(* IEC 61131-3 sources: ironplc-benchmarks/benchmarks/programs, 13 files *)

(* ---- arithmetic.st ---- *)
(* arithmetic.st — Integer arithmetic operations.
   Exercises ADD, SUB, MUL, DIV, and MOD with analytically verifiable
   outputs. After each cycle, result_add = 30, result_sub = 10,
   result_mul = 200, result_div = 2, result_mod = 0. *)

PROGRAM arithmetic
VAR
    a : INT := 20;
    b : INT := 10;
    result_add : INT;
    result_sub : INT;
    result_mul : INT;
    result_div : INT;
    result_mod : INT;
END_VAR
    result_add := a + b;
    result_sub := a - b;
    result_mul := a * b;
    result_div := a / b;
    result_mod := a MOD b;
END_PROGRAM

(* ---- blinky.st ---- *)
(* blinky.st — Minimal benchmark baseline.
   Toggles an output coil on each scan cycle. Exercises the absolute
   minimum VM path: variable read, boolean NOT, variable write. *)

PROGRAM blinky
VAR
    output : BOOL := FALSE;
END_VAR
    output := NOT output;
END_PROGRAM

(* ---- case_state.st ---- *)
(* case_state.st — CASE-based state machine.
   Cycles through 4 states on each scan. Exercises CASE/branch opcodes
   which map to jump tables in both compiled and interpreted execution. *)

PROGRAM case_state
VAR
    state : INT := 0;
    output_a : BOOL := FALSE;
    output_b : BOOL := FALSE;
    output_c : BOOL := FALSE;
    output_d : BOOL := FALSE;
END_VAR
    CASE state OF
        0:
            output_a := TRUE;
            output_b := FALSE;
            output_c := FALSE;
            output_d := FALSE;
            state := 1;
        1:
            output_a := FALSE;
            output_b := TRUE;
            output_c := FALSE;
            output_d := FALSE;
            state := 2;
        2:
            output_a := FALSE;
            output_b := FALSE;
            output_c := TRUE;
            output_d := FALSE;
            state := 3;
        3:
            output_a := FALSE;
            output_b := FALSE;
            output_c := FALSE;
            output_d := TRUE;
            state := 0;
    END_CASE;
END_PROGRAM

(* ---- counter_up.st ---- *)
(* counter_up.st — Counter with reset.
   Exercises integer arithmetic, comparison, and conditional assignment.
   The counter increments each cycle and resets at a threshold. *)

PROGRAM counter_up
VAR
    count : INT := 0;
    threshold : INT := 1000;
    reset_flag : BOOL := FALSE;
END_VAR
    IF count >= threshold THEN
        count := 0;
        reset_flag := TRUE;
    ELSE
        count := count + 1;
        reset_flag := FALSE;
    END_IF;
END_PROGRAM

(* ---- for_loop.st ---- *)
(* for_loop.st — FOR loop with accumulator.
   Exercises loop control flow opcodes. Sums integers 1..100 each cycle,
   producing a verifiable result of 5050. *)

PROGRAM for_loop
VAR
    i : INT;
    total : INT := 0;
END_VAR
    total := 0;
    FOR i := 1 TO 100 DO
        total := total + i;
    END_FOR;
END_PROGRAM

(* ---- oscat_binom.st ---- *)
(* oscat_binom.st — Binomial coefficient from OSCAT library.
   Source: https://github.com/PLC-lang/oscat (OSCAT BASIC, www.oscat.de)
   Exercises: FOR loop, IF/ELSIF/ELSE, RETURN, integer multiply/divide.
   BINOM(10, 5) = 252 each cycle. *)

FUNCTION BINOM : DINT
VAR_INPUT
	N : INT;
	K : INT;
END_VAR
VAR
	i: INT;
END_VAR
(* @END_DECLARATION := '0' *)
IF 2 * K > n THEN
	k := n - k;
END_IF;
IF k > n THEN
	RETURN;
ELSIF k = 0 OR k = n THEN
	BINOM := 1;
ELSIF k = 1 THEN
	BINOM := n;
ELSE
	BINOM := n;
	n := n + 1;
	FOR i := 2 TO k DO
		BINOM := BINOM * (n - i) / i;
	END_FOR;
END_IF;
END_FUNCTION

PROGRAM oscat_binom
VAR
    result : INT;
END_VAR
    result := DINT_TO_INT(BINOM(N := 10, K := 5));
END_PROGRAM

(* ---- oscat_expn.st ---- *)
(* oscat_expn.st — Fast integer exponentiation by squaring from OSCAT.
   Source: https://github.com/PLC-lang/oscat (OSCAT BASIC, www.oscat.de)
   Exercises: WHILE loop, bit access (.0, .15), SHR, REAL arithmetic.
   EXPN(2.0, 10) = 1024.0 each cycle. *)

FUNCTION EXPN : REAL
VAR_INPUT
	X : REAL;
	N : INT;
END_VAR
VAR
	sign: BOOL;
END_VAR
(* @END_DECLARATION := '0' *)
sign := n.15;
N := ABS(N);
IF N.0 THEN EXPN := X; ELSE EXPN := 1.0; END_IF;
N := SHR(N,1);
WHILE N > 0 DO
   X := X * X;
   IF N.0 THEN EXPN := EXPN * X; END_IF;
   N := SHR(N,1);
END_WHILE;
IF sign THEN EXPN := 1.0 / EXPN; END_IF;
END_FUNCTION

PROGRAM oscat_expn
VAR
    result : INT;
END_VAR
    result := REAL_TO_INT(EXPN(X := 2.0, N := 10));
END_PROGRAM

(* ---- oscat_fib.st ---- *)
(* oscat_fib.st — Fibonacci sequence from OSCAT library.
   Source: https://github.com/PLC-lang/oscat (OSCAT BASIC, www.oscat.de)
   Exercises: WHILE loop, IF/ELSIF/ELSE, RETURN, integer arithmetic.
   FIB(20) = 6765 each cycle. *)

FUNCTION FIB : DINT
VAR_INPUT
	X : INT;
END_VAR
VAR
	t1, t2: DINT;
END_VAR
(* @END_DECLARATION := '0' *)
IF X < 0 OR X > 46 THEN
	FIB := -1;
ELSIF x < 2 THEN
	FIB := X;
	RETURN;
ELSE
	t2 := 1;
	WHILE X > 3 DO
		X := X-2;
		t1 := t1 + t2;
		t2 := t1 + t2;
	END_WHILE;
	IF X > 2 THEN t1 := t1 + t2; END_IF;
	fib := t1 + t2;
END_IF;
END_FUNCTION

PROGRAM oscat_fib
VAR
    result : INT;
END_VAR
    result := DINT_TO_INT(FIB(X := 20));
END_PROGRAM

(* ---- oscat_gcd.st ---- *)
(* oscat_gcd.st — Greatest common divisor (Stein's binary algorithm) from OSCAT.
   Source: https://github.com/PLC-lang/oscat (OSCAT BASIC, www.oscat.de)
   Exercises: nested WHILE loops, bit access (.0), SHR/SHL, ABS.
   GCD(48, 36) = 12 each cycle. *)

FUNCTION GCD : INT
VAR_INPUT
	A : DINT;
	B : DINT;
END_VAR
VAR
	t: DINT;
END_VAR
(* @END_DECLARATION := '0' *)
IF A = 0 THEN
	GCD := DINT_TO_INT(ABS(B));
ELSIF B = 0 THEN
	GCD := DINT_TO_INT(ABS(A));
ELSE
	A := ABS(A);
	B := ABS(B);
	GCD := 1;
	WHILE NOT(A.0 OR B.0) DO
		A := SHR(A,1);
		B := SHR(B,1);
		GCD := SHL(GCD,1);
	END_WHILE;
	WHILE A > 0 DO
		IF NOT(A.0) THEN A := SHR(A,1);
		ELSIF NOT(B.0) THEN B := SHR(B,1);
		ELSE
			t:= SHR(ABS(A-B),1);
			IF A < B THEN B := t; ELSE A := T; END_IF;
		END_IF;
	END_WHILE;
	GCD := GCD * DINT_TO_INT(B);
END_IF;
END_FUNCTION

PROGRAM oscat_gcd
VAR
    result : INT;
END_VAR
    result := GCD(A := 48, B := 36);
END_PROGRAM

(* ---- oscat_lambert_w.st ---- *)
(* oscat_lambert_w.st — Lambert W function from OSCAT.
   Source: https://github.com/PLC-lang/oscat (OSCAT BASIC, www.oscat.de)
   Exercises: FOR loop with EXIT, EXP, LN, REAL arithmetic, RETURN,
   IF/ELSIF/ELSE, REAL_TO_DW (bitwise float comparison via REF_TO).
   LAMBERT_W(1.0) ~= 0.5671 each cycle, result = 5671. *)

FUNCTION REAL_TO_DW : DWORD
VAR_INPUT
	X : REAL;
END_VAR
VAR
	pt : REF_TO DWORD;
END_VAR
(* @END_DECLARATION := '0' *)
pt := REF(X);
REAL_TO_DW := pt^;
END_FUNCTION

FUNCTION LAMBERT_W : REAL
VAR_INPUT
	X : REAL;
END_VAR
VAR
	w : REAL;
	i : INT;
	we: REAL;
	w1e: REAL;
	last: DWORD;
	ewx: REAL;
END_VAR
(* @END_DECLARATION := '0' *)
IF x < -0.367879441171442 THEN
	LAMBERT_W := -1000.0;
	RETURN;
ELSIF x = 0.0 THEN
	RETURN;
ELSIF x <= 500.0 THEN
	w := LN(x + 1.0);
	w := 0.665 * (1.0 + 0.0195 * w) * w + 0.04;
ELSE
	w := LN(x - 4.0) - (1.0 - 1.0/LN(x)) * LN(LN(x));
END_IF;
FOR i := 0 TO 5 DO
	ewx := EXP(w);
	we := w * ewx - x;
	w1e := (w+1.0) * ewx;
	last := REAL_TO_DW(w) AND 16#FFFF_FFFC;
	w := w - (we / (w1e - (w+2.0) * we / (2.0 * w + 2.0)));
	IF (REAL_TO_DW(w) AND 16#FFFF_FFFC) = last THEN EXIT; END_IF;
END_FOR;
LAMBERT_W := w;
END_FUNCTION

PROGRAM oscat_lambert_w
VAR
    result : INT;
END_VAR
    result := REAL_TO_INT(LAMBERT_W(X := 1.0) * 10000.0);
END_PROGRAM

(* ---- oscat_linear_int.st ---- *)
(* oscat_linear_int.st — Piecewise linear interpolation from OSCAT.
   Source: https://github.com/PLC-lang/oscat (OSCAT BASIC, www.oscat.de)
   Exercises: WHILE loop, 2D array access, REAL arithmetic, MIN.
   Interpolates X=25 over 5 points: (0,0),(10,100),(20,200),(30,300),(40,400).
   Result = 250 each cycle. *)

FUNCTION LINEAR_INT : REAL
VAR_INPUT
	X : REAL;
	XY : ARRAY[1..20,0..1] OF REAL;
	Pts : INT;
END_VAR
VAR
	i : INT;
END_VAR
(* @END_DECLARATION := '0' *)
pts := MIN(pts,20);

i := 2;
WHILE (i < pts) AND (XY[i,0] < X) DO
	i := i + 1;
END_WHILE;

LINEAR_INT := ((XY[i,1] - XY[i-1,1]) * X - XY[i,1] * XY[i-1,0] + XY[i-1,1] * XY[i,0]) / (XY[i,0] - XY[i-1,0]);
END_FUNCTION

PROGRAM oscat_linear_int
VAR
    points : ARRAY[1..20,0..1] OF REAL;
    result : INT;
END_VAR
    points[1,0] := 0.0;   points[1,1] := 0.0;
    points[2,0] := 10.0;  points[2,1] := 100.0;
    points[3,0] := 20.0;  points[3,1] := 200.0;
    points[4,0] := 30.0;  points[4,1] := 300.0;
    points[5,0] := 40.0;  points[5,1] := 400.0;
    result := REAL_TO_INT(LINEAR_INT(X := 25.0, XY := points, Pts := 5));
END_PROGRAM

(* ---- oscat_polynom_int.st ---- *)
(* oscat_polynom_int.st — Newton polynomial interpolation from OSCAT.
   Source: https://github.com/PLC-lang/oscat (OSCAT BASIC, www.oscat.de)
   Exercises: nested FOR loops (BY -1), 2D array access, REAL arithmetic, MIN.
   Interpolates X=2.5 over y=x^2 points: (1,1),(2,4),(3,9),(4,16),(5,25).
   Result = REAL_TO_INT(6.25) = 6 each cycle. *)

FUNCTION POLYNOM_INT : REAL
VAR_INPUT
	X : REAL;
	XY : ARRAY[1..5,0..1] OF REAL;
	Pts : INT;
END_VAR
VAR
	I, J : INT;
	stop: INT;
END_VAR
(* @END_DECLARATION := '0' *)
pts := MIN(pts, 5);

FOR i := 1 TO pts DO
	stop := i + 1;
   	FOR j := pts TO stop BY -1 DO
   		XY[j,1] := (XY[j,1] - XY[j-1,1]) / (XY[j,0] - XY[j-i,0]);
	END_FOR;
END_FOR;

POLYNOM_INT := 0.0;
FOR i := pts TO 1 BY -1 DO
       POLYNOM_INT := POLYNOM_INT * (X - XY[i,0]) + XY[i,1];
END_FOR;
END_FUNCTION

PROGRAM oscat_polynom_int
VAR
    points : ARRAY[1..5,0..1] OF REAL;
    result : INT;
END_VAR
    points[1,0] := 1.0;  points[1,1] := 1.0;
    points[2,0] := 2.0;  points[2,1] := 4.0;
    points[3,0] := 3.0;  points[3,1] := 9.0;
    points[4,0] := 4.0;  points[4,1] := 16.0;
    points[5,0] := 5.0;  points[5,1] := 25.0;
    result := REAL_TO_INT(POLYNOM_INT(X := 2.5, XY := points, Pts := 5));
END_PROGRAM

(* ---- oscat_real_to_frac.st ---- *)
(* oscat_real_to_frac.st — Real to fraction (continued fractions) from OSCAT.
   Source: https://github.com/PLC-lang/oscat (OSCAT BASIC, www.oscat.de)
   Exercises: REPEAT/UNTIL loop, EXIT, IF/ELSE, REAL/DINT arithmetic,
   struct return type, ABS, type conversions.
   REAL_TO_FRAC(3.14159, 1000) = 355/113 each cycle. *)

TYPE FRACTION :
STRUCT
	NUMERATOR : INT;
	DENOMINATOR : INT;
END_STRUCT
END_TYPE

FUNCTION REAL_TO_FRAC : FRACTION
VAR_INPUT
	X : REAL;
	N : INT;
END_VAR
VAR
	temp : DINT;
	sign: BOOL;
	X_gerundet: DINT;
	X_ohne_Nachkomma: REAL;
	Numerator:       DINT := 1;
	Denominator:     DINT := 0;
	Numerator_old:   DINT := 0;
	Denominator_old: DINT := 1;
END_VAR
(* @END_DECLARATION := '0' *)
IF X < 0.0 THEN
	sign := TRUE;
	X := ABS(X);
END_IF;

REPEAT
	X_gerundet := REAL_TO_DINT(X);

	temp := numerator * X_gerundet + numerator_old;
	numerator_old := numerator;
	numerator := temp;

	temp := denominator * X_gerundet + denominator_old;
	denominator_old := denominator;
	denominator := temp;

	X_ohne_Nachkomma := DINT_TO_REAL(X_gerundet);
	IF X = X_ohne_Nachkomma THEN
		IF ABS(denominator) <= N THEN
			numerator_old := numerator;
			denominator_old := denominator;
		END_IF;
		EXIT;
	ELSE
		X := 1.0 / (X - X_ohne_Nachkomma);
	END_IF;

UNTIL
	ABS(Denominator) > N
END_REPEAT;

IF sign THEN
	REAL_TO_FRAC.NUMERATOR := -1 * ABS(DINT_TO_INT(numerator_old));
ELSE
	REAL_TO_FRAC.NUMERATOR :=  ABS(DINT_TO_INT(numerator_old));
END_IF;
REAL_TO_FRAC.DENOMINATOR := ABS(DINT_TO_INT(denominator_old));
END_FUNCTION

PROGRAM oscat_real_to_frac
VAR
    temp : FRACTION;
    result_num : INT;
    result_den : INT;
END_VAR
    temp := REAL_TO_FRAC(X := 3.14159, N := 1000);
    result_num := temp.NUMERATOR;
    result_den := temp.DENOMINATOR;
END_PROGRAM
